TYPE ST_SafetyScannerSection EXTENDS ST_SectionBase :
STRUCT
END_STRUCT
END_TYPE

(* stored: Version 1.1.0.1, ProductVersion 3.1.4024.12
   DUT ST_SafetyScannerSection: Id {82b897d8-ebe6-4e81-b790-8f2135781d14} *)
